{attribute 'OPC.UA.DA.StructuredType' := '1'}
FUNCTION_BLOCK FB_DosingPumpAgrowtek_R2_1 EXTENDS FB_BaseDevice IMPLEMENTS I_PumpDosing

VAR_IN_OUT
	{attribute 'OPC.UA.DA' := '0'}
	//fbModbusMaster: FB_ModbusMaster;
	fbModbusManager: FB_ModbusManager;
END_VAR

VAR_INPUT
	nModbusUnitID: UINT; 
END_VAR

VAR
	// Modbus Variables
	nPumpID: UINT;	// Pump ID is different to the modbus ID because there are 5 pumps on the 1 modbus address
	 
	ePumpType: E_DosingPump;

	
	bEnableComms: BOOL := TRUE;
	bFirtRun: BOOL := TRUE;
	bResetTimer: BOOL := TRUE;
	
	// Async Statemachine Variables
	{attribute 'OPC.UA.DA' := '0'}
	eSMState: (WAIT, DOSING_TRIG, DOSING, DOSING_OFF_TRIG, DOSED);
	
	// Dosing Variables
	{attribute 'OPC.UA.DA' := '0'} 
	fbTONdoseTime: TON;  
	{attribute 'OPC.UA.DA' := '1'} 
	nDoseRateMLph: UINT;
	{attribute 'OPC.UA.DA' := '1'} 
	nDoseQtyMls: REAL;
	{attribute 'OPC.UA.DA' := '1'} 
	tTimeToDose: TIME;
	
	// delay between writing pump speed and reading pump speed
	fbTONreadDelay : TON := (PT := T#1S);

	// Variables updated over Modbus
	{attribute 'OPC.UA.DA' := '1'} 
	nPumpSpeed_Requested: UINT;
	
	{attribute 'OPC.UA.DA' := '1'} 
	nPumpSpeed: UINT;
	{attribute 'OPC.UA.DA' := '1'} 
	nPumpRunTime: UINT; 
	
	tDataRefresh: TIME := T#10S;
	fbTON_DataRefresh: 	TON := (PT := tDataRefresh, IN := FALSE);
	fbTON_MsgTimeout: 	TON := (PT := T#4S, IN := FALSE);
	
	// Modbus Requests
	stModRead_MotorSpeed: 	ST_Modbus_ReadRequest;
	stModRead_MotorRunTime: ST_Modbus_ReadRequest;
	stModWrite_MotorSpeed: 	ST_Modbus_WriteRequest;
	stModWrite_SetID: 		ST_Modbus_WriteRequest;
	
	
	bRaiseError1: BOOL := FALSE;
	bClearError: BOOL := FALSE;
	bRaiseError2: BOOL := FALSE;
	
	
END_VAR

fbTONdoseTime();
fbTON_MsgTimeout();
fbTON_DataRefresh();
fbTONreadDelay();

IF GVL.bAutoUpdateDeviceState THEN
	eState := eStateTarget;	
END_IF

IF bFirtRun THEN
	init_ModbusRequests();
	bFirtRun := FALSE;
END_IF

IF eMode = E_DeviceMode.MANUAL THEN
	bEnable := TRUE;
END_IF
(*

IF bEnable AND eStateTarget = E_DeviceState.ON AND eState <> E_DeviceState.RUNNING THEN
		eSMState := WAIT;
END_IF

IF (bEnable = FALSE OR eStateTarget = E_DeviceState.IDLE) AND eState <> E_DeviceState.IDLE THEN
		eSMState := 0;
END_IF
*)


IF bResetTimer THEN
	fbTON_DataRefresh.IN := TRUE;
	bResetTimer := FALSE;
END_IF

// Asynchronous update of local variables from the Modbus request structures
nPumpSpeed 		:= WORD_TO_UINT(stModRead_MotorSpeed.ReadRegsVals[1]);
nPumpRunTime 	:= WORD_TO_UINT(stModRead_MotorRunTime.ReadRegsVals[1]);
	
// Request update of local veriables every Xs (in accordance with adjustable DataRefresh timer)
(*IF fbTON_DataRefresh.Q AND bEnable THEN // AND bEnableComms THEN
	// fbModbusManager.addRequest_Read_Priority(ReadRequest := ADR(stModRead_MotorRunTime));
	fbModbusManager.addRequest_Read_Priority(ReadRequest := ADR(stModRead_MotorSpeed));
	fbTON_DataRefresh.IN := FALSE;
	bResetTimer := TRUE;
END_IF
*)


// Statemachine to handle dosing commands
//IF eState = E_Devicestate.RUNNING THEN //AND bEnableComms THEN
	CASE eSMState OF
	
		WAIT:
			// Wait for a dosing command
			eState := E_DeviceState.IDLE;
			// Beau make sure the timeout timer is cleared in case it was left on last time
			fbTON_MsgTimeout.IN := FALSE;
			
		DOSING_TRIG:
			// A call to the 'executeDose' has been received, send modbus command
			// Send the dosing modbus request and start the timer
			//nPumpSpeed_Requested := 100;
			stModWrite_MotorSpeed.WriteRegVals[1] := UINT_TO_WORD(nPumpSpeed_Requested);
			fbModbusManager.addRequest_Write_Priority(WriteRequest := ADR(stModWrite_MotorSpeed));
			// Beau instead of reading pump speed immediately, start the delay timer
			fbTONreadDelay.IN := TRUE;
			//fbModbusManager.addRequest_Read_Priority(ReadRequest := ADR(stModRead_MotorSpeed));
			fbTONdoseTime.IN := TRUE;
			fbTON_MsgTimeout.PT := fbTONdoseTime.PT + T#1S;
			fbTON_MsgTimeout.IN := TRUE;
			eSMState := DOSING;
			eState := E_DeviceState.RUNNING;
			
	
		DOSING: 
		
			// Beau try to read pump speed one second after writing pump speed
			IF fbTONreadDelay.Q THEN
				fbModbusManager.addRequest_Read_Priority(ReadRequest := ADR(stModRead_MotorSpeed));	
				// reset the timer so we don't send another read request
				fbTONreadDelay.IN := FALSE;
			END_IF
			
			IF fbTON_MsgTimeout.Q AND NOT (nPumpSpeed_Requested = nPumpSpeed) THEN
				// The pump hasn't turned on after it was requested to - try again!
				fbModbusManager.addRequest_Read_Priority(ReadRequest := ADR(stModRead_MotorSpeed));
				fbTONdoseTime.IN := FALSE;
				fbTON_MsgTimeout.IN := FALSE;
				eSMState := DOSING_TRIG; // go back and retry
			END_IF
			
			
			IF fbTONdoseTime.Q THEN
				fbTONdoseTime.IN := FALSE; // reset the timer
				IF nPumpSpeed = nPumpSpeed_Requested THEN
					fbTONdoseTime.IN := FALSE;
					fbTON_MsgTimeout.IN := FALSE;
					eSMState := DOSING_OFF_TRIG; // the pump turned on, now we can turn off
				END_IF
			END_IF
			eState := E_DeviceState.RUNNING;
				
			
		DOSING_OFF_TRIG:
			
			// Monitor the run time / compare against the calculated dosing time
			// when dosing time has been exceeded move to dosed
			nPumpSpeed_Requested := 0; // turn the pump off
			stModWrite_MotorSpeed.WriteRegVals[1] := UINT_TO_WORD(nPumpSpeed_Requested);
			
			fbModbusManager.addRequest_Write_Priority(WriteRequest := ADR(stModWrite_MotorSpeed));
			
			fbModbusManager.addRequest_Read_Priority(ReadRequest := ADR(stModRead_MotorSpeed));
			
			fbModbusManager.addRequest_Write_Priority(WriteRequest := ADR(stModWrite_MotorSpeed));
			fbModbusManager.addRequest_Write_Priority(WriteRequest := ADR(stModWrite_MotorSpeed));
			fbModbusManager.addRequest_Write_Priority(WriteRequest := ADR(stModWrite_MotorSpeed));
			fbTON_MsgTimeout.IN := TRUE;
			fbTON_MsgTimeout.PT := T#1s;;
			eSMState := DOSED;
			eState := E_DeviceState.RUNNING;
			
			
		DOSED: 
			// Confirm that the pump has stopped by reading the pump speed 
			// go back to wait if the pump speed has reached 0
			
			IF fbTON_MsgTimeout.Q THEN
				fbTON_MsgTimeout.IN := FALSE;
				IF NOT(nPumpSpeed_Requested = nPumpSpeed) THEN
					// The pump hasn't turned off after it was requested to - try again!
					eSMState := DOSING_OFF_TRIG; // go back and retry
				ELSIF nPumpSpeed_Requested = nPumpSpeed THEN
					eSMState := WAIT; // go back to waiting for the next dose
					nDoseQtyMls := 0; // reset this to 0 for SCADA 
				END_IF
			END_IF
			
			// eSMState := WAIT;
			
	
	END_CASE

//END_IF

{warning 'add method implementation '}
METHOD executeDose : BOOL
VAR_INPUT
	DoseQtyMls: LREAL;
	DoseRateMlph: UINT;
	RequestComplete: 	POINTER TO BOOL;
END_VAR
VAR_OUTPUT
	RequestAccepted: BOOL;
END_VAR
(* setDose dispenses the amount requested at a user requested dose rate *)

//nDoseQtyMls := REAL_TO_UINT((UINT_TO_REAL(DoseQtyMls)/10000.0));
IF (bEnable AND bEnableComms) OR (eMode = E_DeviceMode.MANUAL)  THEN
	// nDoseQtyMls := ABS(DoseQtyMls);

	// IF nDoseQtyMls > 1.0 THEN
	
		nPumpSpeed_Requested := 40;
		//tTimeToDose := REAL_TO_TIME(( nDoseQtyMls / (480.0*(UINT_TO_REAL(nPumpSpeed_Requested)/100.0))) * 60.0 *1000.0);  // Agrowtek maximum flow rate is 480 ml/min
		tTimeToDose := REAL_TO_TIME(( ABS(DoseQtyMls) / (480.0*(UINT_TO_REAL(nPumpSpeed_Requested)/100.0))) * 60.0 *1000.0);  // Agrowtek maximum flow rate is 480 ml/min
		//tTimeToDose := REAL_TO_TIME((((UINT_TO_REAL(nDoseQtyMls)) / 480) * 60.0)*1000);  // Agrowtek maximum flow rate is 480 ml/min
		fbTONdoseTime.PT := tTimeToDose;
	
		IF tTimeToDose >= T#1S THEN
			nDoseQtyMls := ABS(DoseQtyMls);
			eSMState 	:= DOSING_TRIG;
			eState 		:= E_Devicestate.RUNNING;
			bBusy 		:= TRUE;	
		END_IF
	END_IF
END_METHOD

METHOD FB_init : BOOL


VAR_INPUT
	bInitRetains : BOOL; // if TRUE, the retain variables are initialized (warm start / cold start)
	bInCopyCode : BOOL;  // if TRUE, the instance afterwards gets moved into the copy code (online change)
	
	PumpID: STRING;
	PumpDescription: STRING;
	PumpType: E_DosingPump;
	ManifoldModbusID: UINT; 
	
END_VAR
sID := PumpID;
sDescr := PumpDescription;
ePumpType := PumpType;
nModbusUnitID := ManifoldModbusID;
END_METHOD

METHOD getAdrReadAccumRunTime : UINT
VAR_INPUT
	PumpType: E_DosingPump;
END_VAR

VAR
	Address: UINT;
END_VAR
// This method retrieves the Modbus register for the individual Agrowtek pump
// We need to do this because 5 pumps share the same Modbus slave ID, however have differing registers to write to

CASE PumpType OF
	
	E_DosingPump.PH_DOWN:
		Address := 16#64;
		
	E_DosingPump.NUTRIENT_A:
		Address := 16#65;
		
	E_DosingPump.NUTRIENT_B:
		Address := 16#66;

	E_DosingPump.NUTRIENT_C:
		Address := 16#67;
		
	E_DosingPump.PH_UP:
		Address := 16#68;
		
END_CASE

getAdrReadAccumRunTime := Address;
END_METHOD

METHOD getAdrReadWriteSpeed : UINT
VAR_INPUT
	PumpType: E_DosingPump;
END_VAR
// This method retrieves the Modbus register for the individual Agrowtek pump
// We need to do this because 5 pumps share the same Modbus slave ID, however have differing registers to write to

CASE PumpType OF
	
	E_DosingPump.PH_DOWN:
		getAdrReadWriteSpeed := 16#64;
		
	E_DosingPump.NUTRIENT_A:
		getAdrReadWriteSpeed := 16#65;
		
	E_DosingPump.NUTRIENT_B:
		getAdrReadWriteSpeed := 16#66;
		
	E_DosingPump.NUTRIENT_C:
		getAdrReadWriteSpeed := 16#67;
		
	E_DosingPump.PH_UP:
		getAdrReadWriteSpeed := 16#68;
		
END_CASE
END_METHOD

METHOD init_ModbusRequests : BOOL
VAR_INPUT
END_VAR
stModRead_MotorSpeed.SlaveAddress := nModbusUnitID;			
stModRead_MotorSpeed.AdrFirstSlaveRegisterRead := getAdrReadWriteSpeed(PumpType := ePumpType);
stModRead_MotorSpeed.QtyWordsToRead := 1;				// The value is a 16-bit word
stModRead_MotorSpeed.bRequestAccepted := FALSE;
stModRead_MotorSpeed.bRequestCompleted := FALSE;
stModRead_MotorSpeed.ReadRegsVals := GVL.ModbusEmptyBuffer;

stModRead_MotorRunTime.SlaveAddress := nModbusUnitID;			
stModRead_MotorRunTime.AdrFirstSlaveRegisterRead := getAdrReadAccumRunTime(PumpType := ePumpType);
stModRead_MotorRunTime.QtyWordsToRead := 1;				// The value is a 32-bit word
stModRead_MotorRunTime.bRequestAccepted := FALSE;
stModRead_MotorRunTime.bRequestCompleted := FALSE;
stModRead_MotorRunTime.ReadRegsVals := GVL.ModbusEmptyBuffer;


		
stModWrite_MotorSpeed.SlaveAddress := nModbusUnitID;
stModWrite_MotorSpeed.AdrFirstSlaveRegisterWrite := getAdrReadWriteSpeed(PumpType := ePumpType);
stModWrite_MotorSpeed.bRequestAccepted := FALSE;
stModWrite_MotorSpeed.bRequestCompleted := FALSE;
stModWrite_MotorSpeed.QtyWordsToWrite := 1;

stModWrite_SetID.SlaveAddress := 254;
stModWrite_SetID.AdrFirstSlaveRegisterWrite := 0;
stModWrite_SetID.bRequestAccepted := FALSE;
stModWrite_SetID.bRequestCompleted := FALSE;
stModWrite_SetID.QtyWordsToWrite := 1;
END_METHOD

METHOD readSpeed : BOOL
VAR_INPUT
END_VAR
fbModbusManager.addRequest_Read_Priority(ReadRequest := ADR(stModRead_MotorSpeed));
END_METHOD

METHOD setModID : BOOL
VAR_INPUT
	DesiredID: UINT;
END_VAR
stModWrite_SetID.WriteRegVals[1] := DesiredID;
fbModbusManager.addRequest_Write_Priority(WriteRequest := ADR(stModWrite_SetID));
END_METHOD

METHOD setOFF : BOOL
VAR_INPUT
	RequestComplete: 	POINTER TO BOOL;
END_VAR
VAR_OUTPUT
	RequestAccepted: 	BOOL;
END_VAR
eSMState := DOSING_OFF_TRIG;
END_METHOD

METHOD setON : BOOL
VAR_INPUT
	RateMlph	 : 		UINT;
	RequestComplete: 	POINTER TO BOOL;
END_VAR

VAR_OUTPUT
	RequestAccepted: 	BOOL;
END_VAR
END_METHOD

METHOD setSpeed99 : BOOL
VAR_INPUT
END_VAR
nPumpSpeed_Requested := 99;
stModWrite_MotorSpeed.WriteRegVals[1] := UINT_TO_WORD(nPumpSpeed_Requested);
fbModbusManager.addRequest_Write_Priority(WriteRequest := ADR(stModWrite_MotorSpeed));
END_METHOD

END_FUNCTION_BLOCK

(* stored: Version 1.1.0.1, ProductVersion 3.1.4024.12
   POU FB_DosingPumpAgrowtek_R2_1: Id {5ab0e125-d011-43ff-803f-c194f4191e19}, SpecialFunc None
   Method executeDose: Id {7cc8b8eb-b503-4f27-bf92-1e0f263aec54}
   Method FB_init: Id {bf1c6a4f-a8cb-4b92-84e9-5fceeae01f7b}
   Method getAdrReadAccumRunTime: Id {f6fd8bef-6ee3-4d2d-a148-66634fa2c7a8}
   Method getAdrReadWriteSpeed: Id {d745f552-7b1c-410c-9689-c3b14eab1f39}
   Method init_ModbusRequests: Id {bc8a9490-14bc-4420-8e03-20c29716667d}
   Method readSpeed: Id {89747920-f943-4d9d-b609-82e61e4249fa}
   Method setModID: Id {cde2d229-d60b-4e19-b5d1-ed343745cc83}
   Method setOFF: Id {4f1241bf-1735-4243-9d86-514a4270f5bd}
   Method setON: Id {5b4afe73-13f8-469d-99ee-07633d550f54}
   Method setSpeed99: Id {d03b205b-7ae3-4310-89a6-8cb37ca59d21} *)
